(* CoDeSys 2.3 export: LogBufferHandle.EXP *)

(* Data type in core *)
TYPE LogBufferHandle :
STRUCT
    BufferAddress: DWORD;
    BufferSize: DINT;
    BufferEndAddress: DWORD;
    BufferWritePointer: DINT;
    BufferReadPointer: DINT;
    BufferOverflow: DINT;
    MagicByte: BYTE := MAGIC_BYTE_V1_LITTLE_ENDIAN;
END_STRUCT
END_TYPE
